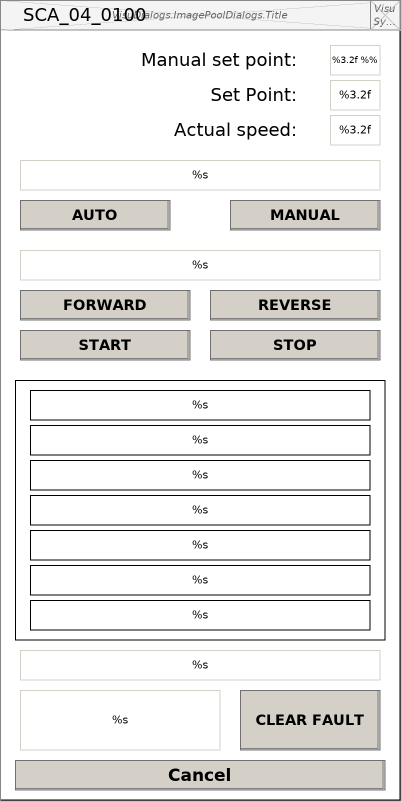
VISUALIZATION visuSCADiag  // 402x802
    Rectangle (0,0 400x800)
    Button (20,200 150x30), "AUTO"
        tap progSCACntrl.SCA_04_0100.AutoReq
    Button (230,200 150x30), "MANUAL"
        tap progSCACntrl.SCA_04_0100.ManReq
    Button (20,290 170x30), "FORWARD"
        OnMouseClick: execute { progSCACntrl.SCA_04_0100.ManDirection := 0; }
    Button (210,290 170x30), "REVERSE"
        OnMouseClick: execute { progSCACntrl.SCA_04_0100.ManDirection := 1; }
    Textfield (20,160 360x30), "%s", text variable: progSCACntrl.SCA_04_0100.strAutoMan
    Textfield (20,250 360x30), "%s", text variable: progSCACntrl.SCA_04_0100.strStopTravRun
    Image (0,0 400x30), image: VisuDialogs.ImagePoolDialogs.Title
    Group (370,0 30x30)
        RoundedRectangle (0,0 30x30)
        Image (0,0 30x30), image: VisuSymbols.Symbols.Wrong
    Rectangle (15,380 370x260)
    RoundedRectangle (30,390 340x30), "%s", text variable: progSCACntrl.SCA_04_0100.strInterlock_1
    RoundedRectangle (30,425 340x30), "%s", text variable: progSCACntrl.SCA_04_0100.strInterlock_2
    RoundedRectangle (30,460 340x30), "%s", text variable: progSCACntrl.SCA_04_0100.strInterlock_3
    RoundedRectangle (30,495 340x30), "%s", text variable: progSCACntrl.SCA_04_0100.strInterlock_4
    RoundedRectangle (30,530 340x30), "%s", text variable: progSCACntrl.SCA_04_0100.strInterlock_5
    RoundedRectangle (30,565 340x30), "%s", text variable: progSCACntrl.SCA_04_0100.strInterlock_6
    RoundedRectangle (30,600 340x30), "%s", text variable: progSCACntrl.SCA_04_0100.strInterlock_7
    Button (15,760 370x30), "Cancel"
    Label (0,80 300x30), "Set Point:"
    Textfield (330,80 50x30), "%3.2f", text variable: progSCACntrl.SCA_04_0100.CommandSpeed
    Label (0,45 300x30), "Manual set point:"
    Textfield (330,45 50x30), "%3.2f %%", text variable: progSCACntrl.SCA_04_0100.ManSpeed
        OnMouseClick: write the text variable via VisuDialogs.Numpad, min progSCACntrl.SCA_04_0100.EngMin, max progSCACntrl.SCA_04_0100.EngMax, format %3.2f
    Label (0,115 300x30), "Actual speed:"
    Textfield (330,115 50x30), "%3.2f", text variable: progSCACntrl.SCA_04_0100.ActualSpeed
    Label (20,0 210x30), "SCA_04_0100"
    Button (20,330 170x30), "START"
        tap progSCACntrl.SCA_04_0100.ManStart
    Button (210,330 170x30), "STOP"
        tap progSCACntrl.SCA_04_0100.ManStop
    Textfield (20,650 360x30), "%s", text variable: progSCACntrl.SCA_04_0100.strAlmDesc
    Textfield (20,690 200x60), "%s", text variable: progSCACntrl.SCA_04_0100.strOKFault
    Button (240,690 140x60), "CLEAR FAULT"
        tap progSCACntrl.SCA_04_0100.ClearFlt
END_VISUALIZATION

(* stored: Version 1.1.0.1, ProductVersion 3.1.4022.17
   Visu visuSCADiag: Id {da2477d1-854b-44fd-b15e-69a58fe7281d} *)
